// TIA Portal V18 export
FUNCTION "Controls" : Void   // FC8, LAD
{ S7_Optimized_Access := 'TRUE' }
VERSION : 0.1
// stored: AutoNumber true, IsIECCheckEnabled false, SetENOAutomatically false, UDAEnableTagReadback false
BEGIN

REGION Network 1: Function selected
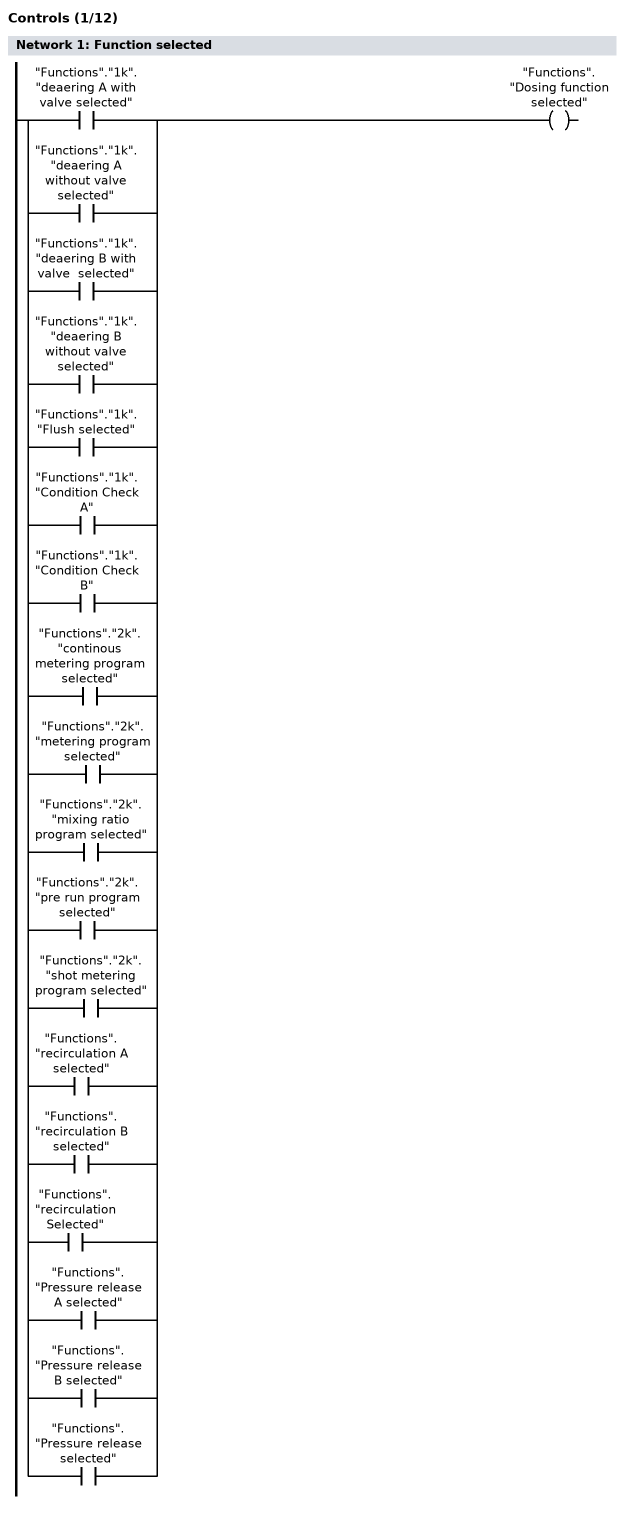
   RUNG wire#powerrail
      Contact( "Functions"."1k"."deaering A with valve selected" )
      wire#w1
      Coil( "Functions"."Dosing function selected" )
   END_RUNG
   RUNG wire#powerrail
      Contact( "Functions"."1k"."deaering A without valve selected" )
   END_RUNG wire#w1
   RUNG wire#powerrail
      Contact( "Functions"."1k"."deaering B with valve  selected" )
   END_RUNG wire#w1
   RUNG wire#powerrail
      Contact( "Functions"."1k"."deaering B without valve  selected" )
   END_RUNG wire#w1
   RUNG wire#powerrail
      Contact( "Functions"."1k"."Flush selected" )
   END_RUNG wire#w1
   RUNG wire#powerrail
      Contact( "Functions"."1k"."Condition Check A" )
   END_RUNG wire#w1
   RUNG wire#powerrail
      Contact( "Functions"."1k"."Condition Check B" )
   END_RUNG wire#w1
   RUNG wire#powerrail
      Contact( "Functions"."2k"."continous metering program selected" )
   END_RUNG wire#w1
   RUNG wire#powerrail
      Contact( "Functions"."2k"."metering program selected" )
   END_RUNG wire#w1
   RUNG wire#powerrail
      Contact( "Functions"."2k"."mixing ratio program selected" )
   END_RUNG wire#w1
   RUNG wire#powerrail
      Contact( "Functions"."2k"."pre run program selected" )
   END_RUNG wire#w1
   RUNG wire#powerrail
      Contact( "Functions"."2k"."shot metering program selected" )
   END_RUNG wire#w1
   RUNG wire#powerrail
      Contact( "Functions"."recirculation A selected" )
   END_RUNG wire#w1
   RUNG wire#powerrail
      Contact( "Functions"."recirculation B selected" )
   END_RUNG wire#w1
   RUNG wire#powerrail
      Contact( "Functions"."recirculation Selected" )
   END_RUNG wire#w1
   RUNG wire#powerrail
      Contact( "Functions"."Pressure release A selected" )
   END_RUNG wire#w1
   RUNG wire#powerrail
      Contact( "Functions"."Pressure release B selected" )
   END_RUNG wire#w1
   RUNG wire#powerrail
      Contact( "Functions"."Pressure release selected" )
   END_RUNG wire#w1
   // the same network as SCL:
   "Functions"."Dosing function selected" := "Functions"."1k"."deaering A with valve selected" OR "Functions"."1k"."deaering A without valve selected" OR "Functions"."1k"."deaering B with valve  selected" OR "Functions"."1k"."deaering B without valve  selected" OR "Functions"."1k"."Flush selected" OR "Functions"."1k"."Condition Check A" OR "Functions"."1k"."Condition Check B" OR "Functions"."2k"."continous metering program selected" OR "Functions"."2k"."metering program selected" OR "Functions"."2k"."mixing ratio program selected" OR "Functions"."2k"."pre run program selected" OR "Functions"."2k"."shot metering program selected" OR "Functions"."recirculation A selected" OR "Functions"."recirculation B selected" OR "Functions"."recirculation Selected" OR "Functions"."Pressure release A selected" OR "Functions"."Pressure release B selected" OR "Functions"."Pressure release selected";
END_REGION

REGION Network 2: Deselect all function
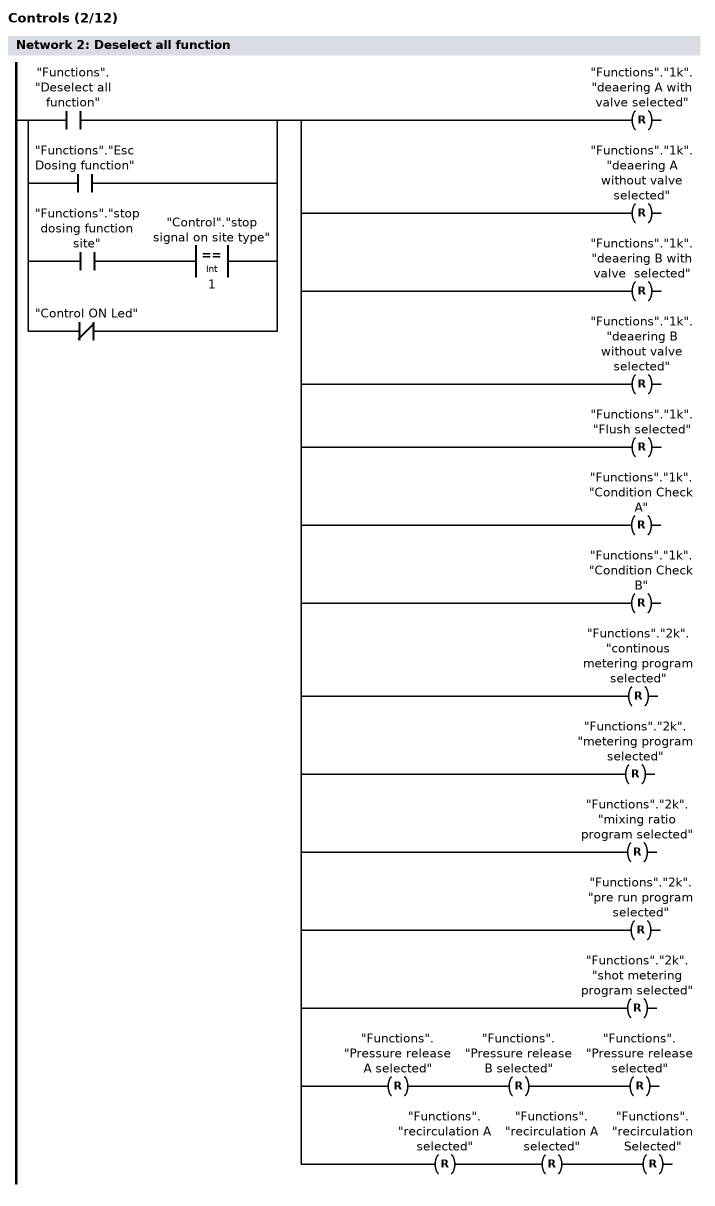
   RUNG wire#powerrail
      Contact( "Functions"."Deselect all function" )
      wire#w1
      R_Coil( "Functions"."1k"."deaering A with valve selected" )
   END_RUNG
   RUNG wire#powerrail
      Contact( "Functions"."Esc Dosing function" )
   END_RUNG wire#w1
   RUNG wire#powerrail
      Contact( "Functions"."stop dosing function site" )
      { S7_Templates := "SrcType := Int" } EQ_Contact(in1 := "Control"."stop signal on site type", in2 := 1)
   END_RUNG wire#w1
   RUNG wire#powerrail
      I_Contact( "Control ON Led" )
   END_RUNG wire#w1
   RUNG wire#w1
      R_Coil( "Functions"."1k"."deaering A without valve selected" )
   END_RUNG
   RUNG wire#w1
      R_Coil( "Functions"."1k"."deaering B with valve  selected" )
   END_RUNG
   RUNG wire#w1
      R_Coil( "Functions"."1k"."deaering B without valve  selected" )
   END_RUNG
   RUNG wire#w1
      R_Coil( "Functions"."1k"."Flush selected" )
   END_RUNG
   RUNG wire#w1
      R_Coil( "Functions"."1k"."Condition Check A" )
   END_RUNG
   RUNG wire#w1
      R_Coil( "Functions"."1k"."Condition Check B" )
   END_RUNG
   RUNG wire#w1
      R_Coil( "Functions"."2k"."continous metering program selected" )
   END_RUNG
   RUNG wire#w1
      R_Coil( "Functions"."2k"."metering program selected" )
   END_RUNG
   RUNG wire#w1
      R_Coil( "Functions"."2k"."mixing ratio program selected" )
   END_RUNG
   RUNG wire#w1
      R_Coil( "Functions"."2k"."pre run program selected" )
   END_RUNG
   RUNG wire#w1
      R_Coil( "Functions"."2k"."shot metering program selected" )
   END_RUNG
   RUNG wire#w1
      R_Coil( "Functions"."Pressure release A selected" )
      R_Coil( "Functions"."Pressure release B selected" )
      R_Coil( "Functions"."Pressure release selected" )
   END_RUNG
   RUNG wire#w1
      R_Coil( "Functions"."recirculation A selected" )
      R_Coil( "Functions"."recirculation A selected" )
      R_Coil( "Functions"."recirculation Selected" )
   END_RUNG
   // the same network as SCL:
   IF "Functions"."Deselect all function" OR "Functions"."Esc Dosing function" OR ("Functions"."stop dosing function site" AND ("Control"."stop signal on site type" = 1)) OR NOT "Control ON Led" THEN
       "Functions"."1k"."deaering A with valve selected" := FALSE;
       "Functions"."1k"."deaering A without valve selected" := FALSE;
       "Functions"."1k"."deaering B with valve  selected" := FALSE;
       "Functions"."1k"."deaering B without valve  selected" := FALSE;
       "Functions"."1k"."Flush selected" := FALSE;
       "Functions"."1k"."Condition Check A" := FALSE;
       "Functions"."1k"."Condition Check B" := FALSE;
       "Functions"."2k"."continous metering program selected" := FALSE;
       "Functions"."2k"."metering program selected" := FALSE;
       "Functions"."2k"."mixing ratio program selected" := FALSE;
       "Functions"."2k"."pre run program selected" := FALSE;
       "Functions"."2k"."shot metering program selected" := FALSE;
       "Functions"."Pressure release A selected" := FALSE;
       "Functions"."Pressure release B selected" := FALSE;
       "Functions"."Pressure release selected" := FALSE;
       "Functions"."recirculation A selected" := FALSE;
       "Functions"."recirculation A selected" := FALSE;
       "Functions"."recirculation Selected" := FALSE;
   END_IF;
END_REGION

REGION Network 3: Deselect all function During Refilling
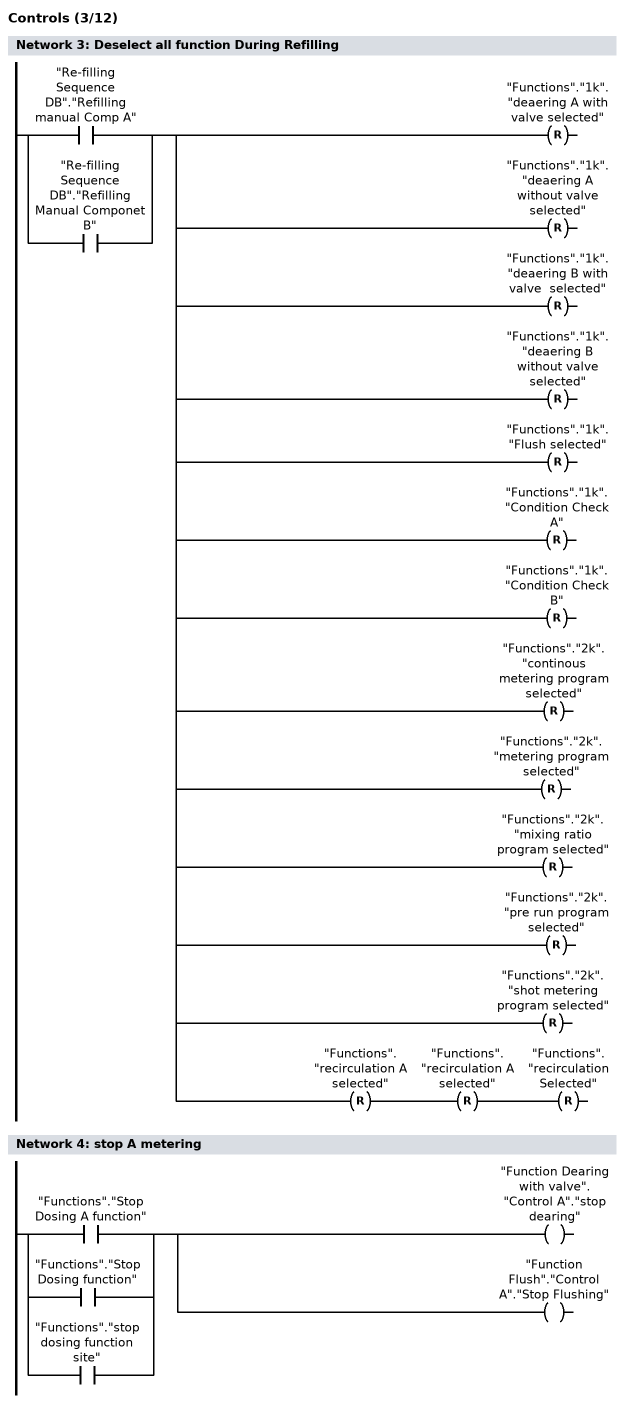
   RUNG wire#powerrail
      Contact( "Re-filling Sequence DB"."Refilling manual Comp A" )
      wire#w1
      R_Coil( "Functions"."1k"."deaering A with valve selected" )
   END_RUNG
   RUNG wire#powerrail
      Contact( "Re-filling Sequence DB"."Refilling Manual Componet B" )
   END_RUNG wire#w1
   RUNG wire#w1
      R_Coil( "Functions"."1k"."deaering A without valve selected" )
   END_RUNG
   RUNG wire#w1
      R_Coil( "Functions"."1k"."deaering B with valve  selected" )
   END_RUNG
   RUNG wire#w1
      R_Coil( "Functions"."1k"."deaering B without valve  selected" )
   END_RUNG
   RUNG wire#w1
      R_Coil( "Functions"."1k"."Flush selected" )
   END_RUNG
   RUNG wire#w1
      R_Coil( "Functions"."1k"."Condition Check A" )
   END_RUNG
   RUNG wire#w1
      R_Coil( "Functions"."1k"."Condition Check B" )
   END_RUNG
   RUNG wire#w1
      R_Coil( "Functions"."2k"."continous metering program selected" )
   END_RUNG
   RUNG wire#w1
      R_Coil( "Functions"."2k"."metering program selected" )
   END_RUNG
   RUNG wire#w1
      R_Coil( "Functions"."2k"."mixing ratio program selected" )
   END_RUNG
   RUNG wire#w1
      R_Coil( "Functions"."2k"."pre run program selected" )
   END_RUNG
   RUNG wire#w1
      R_Coil( "Functions"."2k"."shot metering program selected" )
   END_RUNG
   RUNG wire#w1
      R_Coil( "Functions"."recirculation A selected" )
      R_Coil( "Functions"."recirculation A selected" )
      R_Coil( "Functions"."recirculation Selected" )
   END_RUNG
   // the same network as SCL:
   IF "Re-filling Sequence DB"."Refilling manual Comp A" OR "Re-filling Sequence DB"."Refilling Manual Componet B" THEN
       "Functions"."1k"."deaering A with valve selected" := FALSE;
       "Functions"."1k"."deaering A without valve selected" := FALSE;
       "Functions"."1k"."deaering B with valve  selected" := FALSE;
       "Functions"."1k"."deaering B without valve  selected" := FALSE;
       "Functions"."1k"."Flush selected" := FALSE;
       "Functions"."1k"."Condition Check A" := FALSE;
       "Functions"."1k"."Condition Check B" := FALSE;
       "Functions"."2k"."continous metering program selected" := FALSE;
       "Functions"."2k"."metering program selected" := FALSE;
       "Functions"."2k"."mixing ratio program selected" := FALSE;
       "Functions"."2k"."pre run program selected" := FALSE;
       "Functions"."2k"."shot metering program selected" := FALSE;
       "Functions"."recirculation A selected" := FALSE;
       "Functions"."recirculation A selected" := FALSE;
       "Functions"."recirculation Selected" := FALSE;
   END_IF;
END_REGION

REGION Network 4: stop A metering
   RUNG wire#powerrail
      Contact( "Functions"."Stop Dosing A function" )
      wire#w1
      Coil( "Function Dearing with valve"."Control A"."stop dearing" )
   END_RUNG
   RUNG wire#powerrail
      Contact( "Functions"."Stop Dosing function" )
   END_RUNG wire#w1
   RUNG wire#powerrail
      Contact( "Functions"."stop dosing function site" )
   END_RUNG wire#w1
   RUNG wire#w1
      Coil( "Function Flush"."Control A"."Stop Flushing" )
   END_RUNG
   // the same network as SCL:
   "Function Dearing with valve"."Control A"."stop dearing" := "Functions"."Stop Dosing A function" OR "Functions"."Stop Dosing function" OR "Functions"."stop dosing function site";
   "Function Flush"."Control A"."Stop Flushing" := "Function Dearing with valve"."Control A"."stop dearing";
END_REGION

REGION Network 5: stop B metering
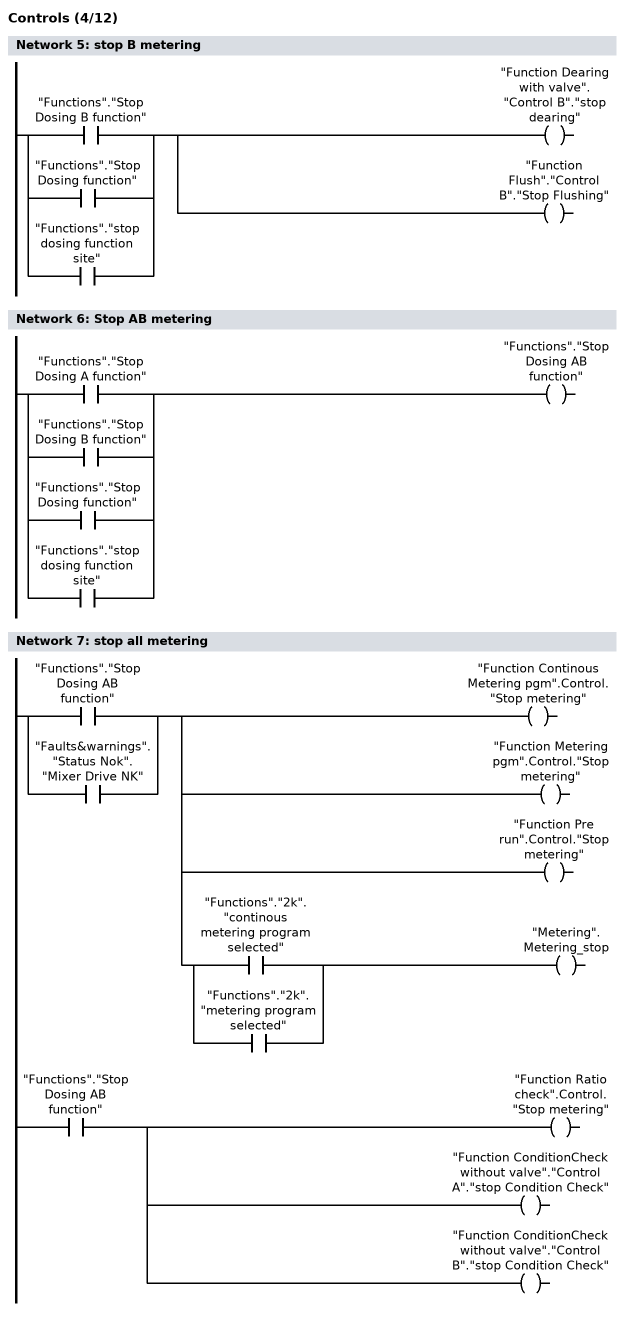
   RUNG wire#powerrail
      Contact( "Functions"."Stop Dosing B function" )
      wire#w1
      Coil( "Function Dearing with valve"."Control B"."stop dearing" )
   END_RUNG
   RUNG wire#powerrail
      Contact( "Functions"."Stop Dosing function" )
   END_RUNG wire#w1
   RUNG wire#powerrail
      Contact( "Functions"."stop dosing function site" )
   END_RUNG wire#w1
   RUNG wire#w1
      Coil( "Function Flush"."Control B"."Stop Flushing" )
   END_RUNG
   // the same network as SCL:
   "Function Dearing with valve"."Control B"."stop dearing" := "Functions"."Stop Dosing B function" OR "Functions"."Stop Dosing function" OR "Functions"."stop dosing function site";
   "Function Flush"."Control B"."Stop Flushing" := "Function Dearing with valve"."Control B"."stop dearing";
END_REGION

REGION Network 6: Stop AB metering
   RUNG wire#powerrail
      Contact( "Functions"."Stop Dosing A function" )
      wire#w1
      Coil( "Functions"."Stop Dosing AB function" )
   END_RUNG
   RUNG wire#powerrail
      Contact( "Functions"."Stop Dosing B function" )
   END_RUNG wire#w1
   RUNG wire#powerrail
      Contact( "Functions"."Stop Dosing function" )
   END_RUNG wire#w1
   RUNG wire#powerrail
      Contact( "Functions"."stop dosing function site" )
   END_RUNG wire#w1
   // the same network as SCL:
   "Functions"."Stop Dosing AB function" := "Functions"."Stop Dosing A function" OR "Functions"."Stop Dosing B function" OR "Functions"."Stop Dosing function" OR "Functions"."stop dosing function site";
END_REGION

REGION Network 7: stop all metering
   RUNG wire#powerrail
      Contact( "Functions"."Stop Dosing AB function" )
      wire#w1
      Coil( "Function Continous Metering pgm".Control."Stop metering" )
   END_RUNG
   RUNG wire#powerrail
      Contact( "Faults&warnings"."Status Nok"."Mixer Drive NK" )
   END_RUNG wire#w1
   RUNG wire#w1
      Coil( "Function Metering pgm".Control."Stop metering" )
   END_RUNG
   RUNG wire#w1
      Coil( "Function Pre run".Control."Stop metering" )
   END_RUNG
   RUNG wire#w1
      Contact( "Functions"."2k"."continous metering program selected" )
      wire#w2
      Coil( "Metering".Metering_stop )
   END_RUNG
   RUNG wire#w1
      Contact( "Functions"."2k"."metering program selected" )
   END_RUNG wire#w2
   RUNG wire#powerrail
      Contact( "Functions"."Stop Dosing AB function" )
      wire#w3
      Coil( "Function Ratio check".Control."Stop metering" )
   END_RUNG
   RUNG wire#w3
      Coil( "Function ConditionCheck without valve"."Control A"."stop Condition Check" )
   END_RUNG
   RUNG wire#w3
      Coil( "Function ConditionCheck without valve"."Control B"."stop Condition Check" )
   END_RUNG
   // the same network as SCL:
   "Function Continous Metering pgm".Control."Stop metering" := "Functions"."Stop Dosing AB function" OR "Faults&warnings"."Status Nok"."Mixer Drive NK";
   "Function Metering pgm".Control."Stop metering" := "Function Continous Metering pgm".Control."Stop metering";
   "Function Pre run".Control."Stop metering" := "Function Continous Metering pgm".Control."Stop metering";
   "Metering".Metering_stop := "Function Continous Metering pgm".Control."Stop metering" AND ("Functions"."2k"."continous metering program selected" OR "Functions"."2k"."metering program selected");
   "Function Ratio check".Control."Stop metering" := "Functions"."Stop Dosing AB function";
   "Function ConditionCheck without valve"."Control A"."stop Condition Check" := "Functions"."Stop Dosing AB function";
   "Function ConditionCheck without valve"."Control B"."stop Condition Check" := "Functions"."Stop Dosing AB function";
END_REGION

REGION Network 8: Critical fault Block A metering
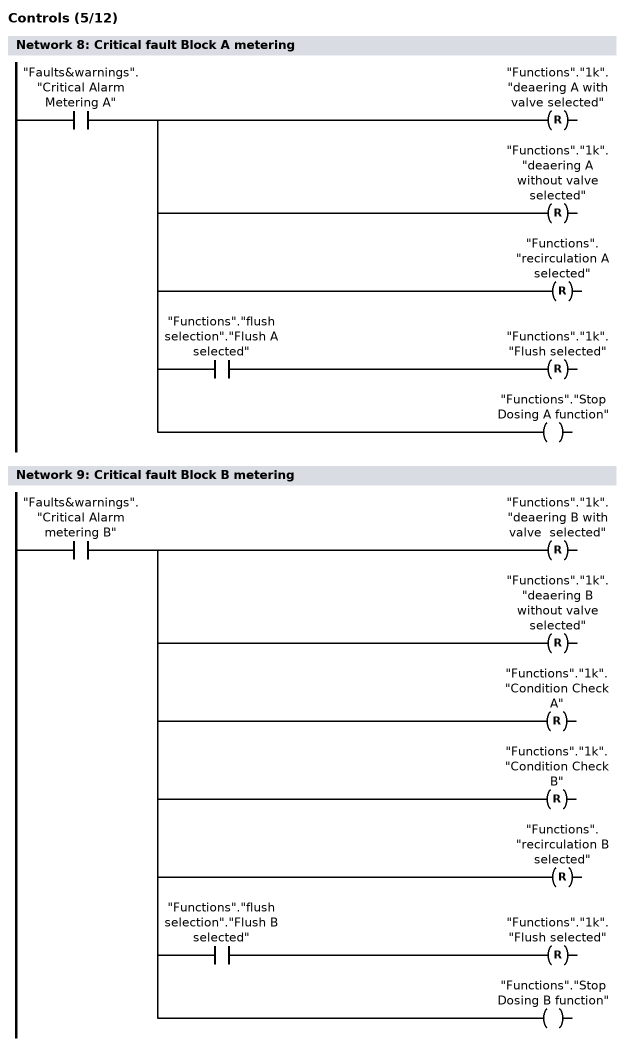
   RUNG wire#powerrail
      Contact( "Faults&warnings"."Critical Alarm Metering A" )
      wire#w1
      R_Coil( "Functions"."1k"."deaering A with valve selected" )
   END_RUNG
   RUNG wire#w1
      R_Coil( "Functions"."1k"."deaering A without valve selected" )
   END_RUNG
   RUNG wire#w1
      R_Coil( "Functions"."recirculation A selected" )
   END_RUNG
   RUNG wire#w1
      Contact( "Functions"."flush selection"."Flush A selected" )
      R_Coil( "Functions"."1k"."Flush selected" )
   END_RUNG
   RUNG wire#w1
      Coil( "Functions"."Stop Dosing A function" )
   END_RUNG
   // the same network as SCL:
   IF "Faults&warnings"."Critical Alarm Metering A" THEN
       "Functions"."1k"."deaering A with valve selected" := FALSE;
       "Functions"."1k"."deaering A without valve selected" := FALSE;
       "Functions"."recirculation A selected" := FALSE;
   END_IF;
   IF "Faults&warnings"."Critical Alarm Metering A" AND "Functions"."flush selection"."Flush A selected" THEN
       "Functions"."1k"."Flush selected" := FALSE;
   END_IF;
   "Functions"."Stop Dosing A function" := "Faults&warnings"."Critical Alarm Metering A";
END_REGION

REGION Network 9: Critical fault Block B metering
   RUNG wire#powerrail
      Contact( "Faults&warnings"."Critical Alarm metering B" )
      wire#w1
      R_Coil( "Functions"."1k"."deaering B with valve  selected" )
   END_RUNG
   RUNG wire#w1
      R_Coil( "Functions"."1k"."deaering B without valve  selected" )
   END_RUNG
   RUNG wire#w1
      R_Coil( "Functions"."1k"."Condition Check A" )
   END_RUNG
   RUNG wire#w1
      R_Coil( "Functions"."1k"."Condition Check B" )
   END_RUNG
   RUNG wire#w1
      R_Coil( "Functions"."recirculation B selected" )
   END_RUNG
   RUNG wire#w1
      Contact( "Functions"."flush selection"."Flush B selected" )
      R_Coil( "Functions"."1k"."Flush selected" )
   END_RUNG
   RUNG wire#w1
      Coil( "Functions"."Stop Dosing B function" )
   END_RUNG
   // the same network as SCL:
   IF "Faults&warnings"."Critical Alarm metering B" THEN
       "Functions"."1k"."deaering B with valve  selected" := FALSE;
       "Functions"."1k"."deaering B without valve  selected" := FALSE;
       "Functions"."1k"."Condition Check A" := FALSE;
       "Functions"."1k"."Condition Check B" := FALSE;
       "Functions"."recirculation B selected" := FALSE;
   END_IF;
   IF "Faults&warnings"."Critical Alarm metering B" AND "Functions"."flush selection"."Flush B selected" THEN
       "Functions"."1k"."Flush selected" := FALSE;
   END_IF;
   "Functions"."Stop Dosing B function" := "Faults&warnings"."Critical Alarm metering B";
END_REGION

REGION Network 10: Critical fault block all metering
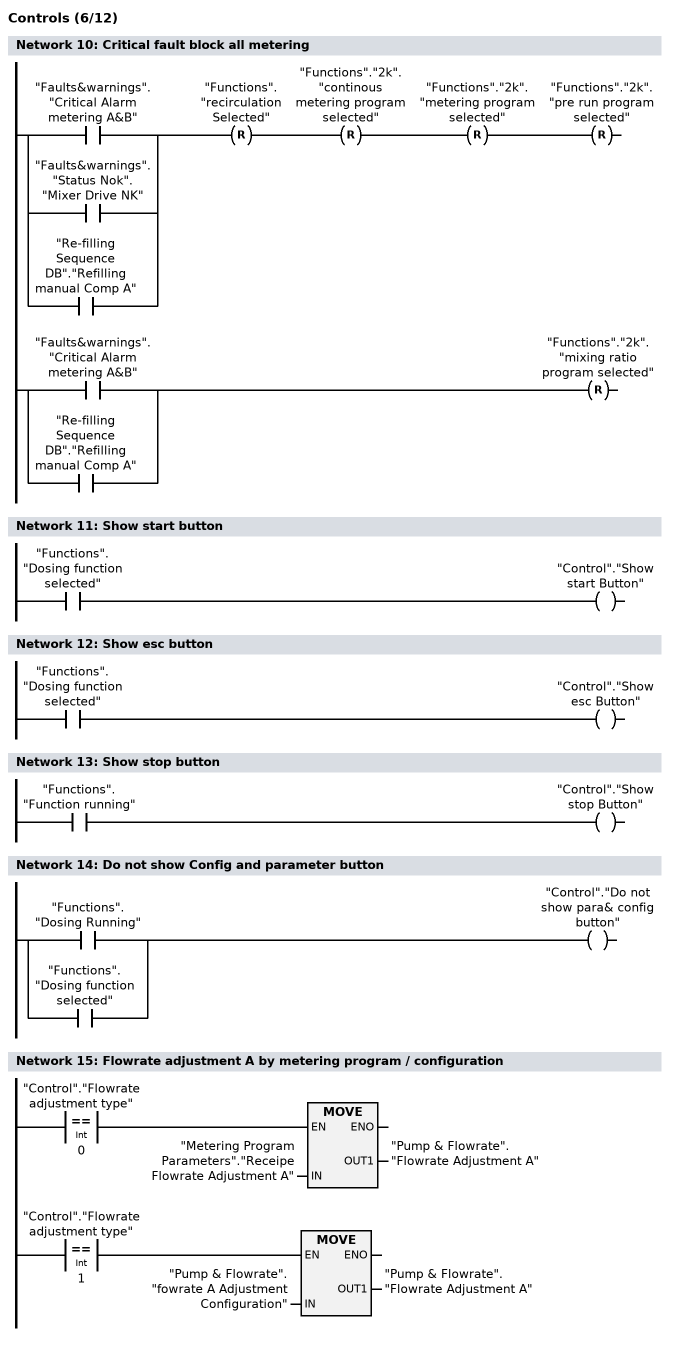
   RUNG wire#powerrail
      Contact( "Faults&warnings"."Critical Alarm metering A&B" )
      wire#w1
      R_Coil( "Functions"."recirculation Selected" )
      R_Coil( "Functions"."2k"."continous metering program selected" )
      R_Coil( "Functions"."2k"."metering program selected" )
      R_Coil( "Functions"."2k"."pre run program selected" )
   END_RUNG
   RUNG wire#powerrail
      Contact( "Faults&warnings"."Status Nok"."Mixer Drive NK" )
   END_RUNG wire#w1
   RUNG wire#powerrail
      Contact( "Re-filling Sequence DB"."Refilling manual Comp A" )
   END_RUNG wire#w1
   RUNG wire#powerrail
      Contact( "Faults&warnings"."Critical Alarm metering A&B" )
      wire#w2
      R_Coil( "Functions"."2k"."mixing ratio program selected" )
   END_RUNG
   RUNG wire#powerrail
      Contact( "Re-filling Sequence DB"."Refilling manual Comp A" )
   END_RUNG wire#w2
   // the same network as SCL:
   IF "Faults&warnings"."Critical Alarm metering A&B" OR "Faults&warnings"."Status Nok"."Mixer Drive NK" OR "Re-filling Sequence DB"."Refilling manual Comp A" THEN
       "Functions"."recirculation Selected" := FALSE;
       "Functions"."2k"."continous metering program selected" := FALSE;
       "Functions"."2k"."metering program selected" := FALSE;
       "Functions"."2k"."pre run program selected" := FALSE;
   END_IF;
   IF "Faults&warnings"."Critical Alarm metering A&B" OR "Re-filling Sequence DB"."Refilling manual Comp A" THEN
       "Functions"."2k"."mixing ratio program selected" := FALSE;
   END_IF;
END_REGION

REGION Network 11: Show start button
   RUNG wire#powerrail
      Contact( "Functions"."Dosing function selected" )
      Coil( "Control"."Show start Button" )
   END_RUNG
   // the same network as SCL:
   "Control"."Show start Button" := "Functions"."Dosing function selected";
END_REGION

REGION Network 12: Show esc button
   RUNG wire#powerrail
      Contact( "Functions"."Dosing function selected" )
      Coil( "Control"."Show esc Button" )
   END_RUNG
   // the same network as SCL:
   "Control"."Show esc Button" := "Functions"."Dosing function selected";
END_REGION

REGION Network 13: Show stop button
   RUNG wire#powerrail
      Contact( "Functions"."Function running" )
      Coil( "Control"."Show stop Button" )
   END_RUNG
   // the same network as SCL:
   "Control"."Show stop Button" := "Functions"."Function running";
END_REGION

REGION Network 14: Do not show Config and parameter button
   RUNG wire#powerrail
      Contact( "Functions"."Dosing Running" )
      wire#w1
      Coil( "Control"."Do not show para& config button" )
   END_RUNG
   RUNG wire#powerrail
      Contact( "Functions"."Dosing function selected" )
   END_RUNG wire#w1
   // the same network as SCL:
   "Control"."Do not show para& config button" := "Functions"."Dosing Running" OR "Functions"."Dosing function selected";
END_REGION

REGION Network 15: Flowrate adjustment A by metering program / configuration
   IF "Control"."Flowrate adjustment type" = 0 THEN
       "Pump & Flowrate"."Flowrate Adjustment A" := "Metering Program Parameters"."Receipe Flowrate Adjustment A";
   END_IF;
   IF "Control"."Flowrate adjustment type" = 1 THEN
       "Pump & Flowrate"."Flowrate Adjustment A" := "Pump & Flowrate"."fowrate A Adjustment Configuration";
   END_IF;
END_REGION

REGION Network 16: Flowrate adjustment B by metering program / configuration
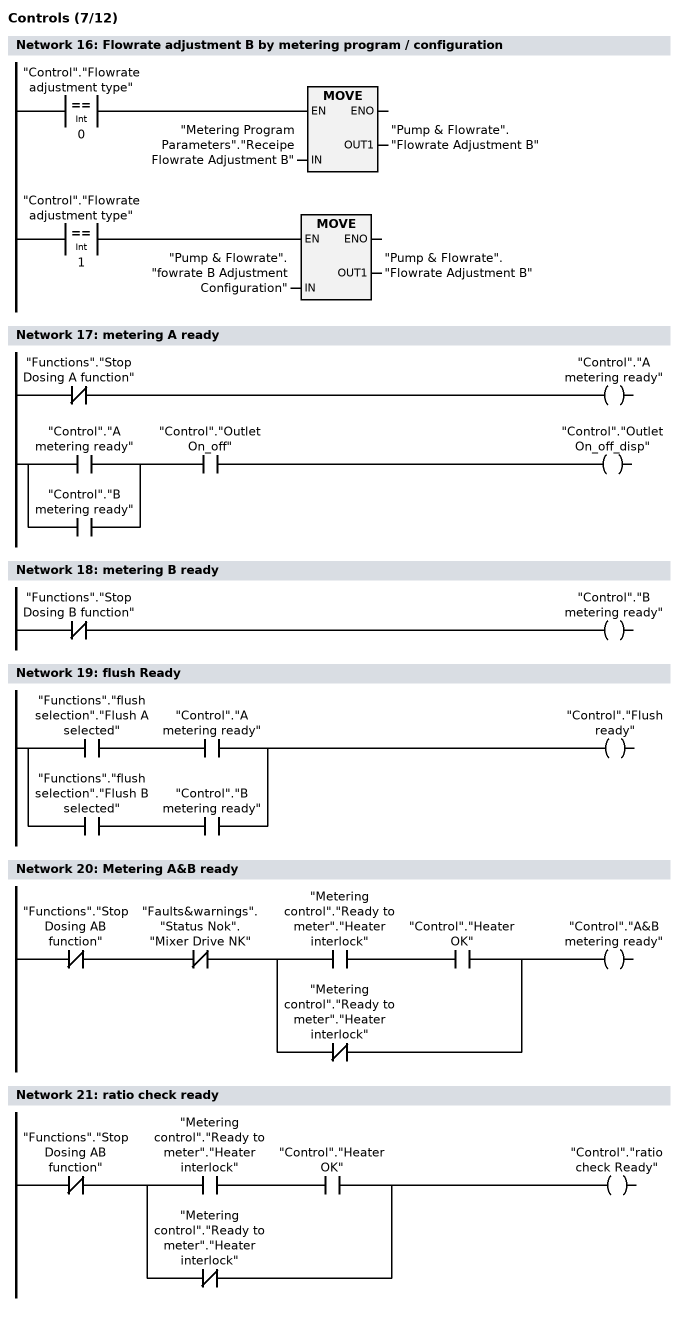
   IF "Control"."Flowrate adjustment type" = 0 THEN
       "Pump & Flowrate"."Flowrate Adjustment B" := "Metering Program Parameters"."Receipe Flowrate Adjustment B";
   END_IF;
   IF "Control"."Flowrate adjustment type" = 1 THEN
       "Pump & Flowrate"."Flowrate Adjustment B" := "Pump & Flowrate"."fowrate B Adjustment Configuration";
   END_IF;
END_REGION

REGION Network 17: metering A ready
   RUNG wire#powerrail
      I_Contact( "Functions"."Stop Dosing A function" )
      Coil( "Control"."A metering ready" )
   END_RUNG
   RUNG wire#powerrail
      Contact( "Control"."A metering ready" )
      wire#w1
      Contact( "Control"."Outlet On_off" )
      Coil( "Control"."Outlet On_off_disp" )
   END_RUNG
   RUNG wire#powerrail
      Contact( "Control"."B metering ready" )
   END_RUNG wire#w1
   // the same network as SCL:
   "Control"."A metering ready" := NOT "Functions"."Stop Dosing A function";
   "Control"."Outlet On_off_disp" := ("Control"."A metering ready" OR "Control"."B metering ready") AND "Control"."Outlet On_off";
END_REGION

REGION Network 18: metering B ready
   RUNG wire#powerrail
      I_Contact( "Functions"."Stop Dosing B function" )
      Coil( "Control"."B metering ready" )
   END_RUNG
   // the same network as SCL:
   "Control"."B metering ready" := NOT "Functions"."Stop Dosing B function";
END_REGION

REGION Network 19: flush Ready
   RUNG wire#powerrail
      Contact( "Functions"."flush selection"."Flush A selected" )
      Contact( "Control"."A metering ready" )
      wire#w1
      Coil( "Control"."Flush ready" )
   END_RUNG
   RUNG wire#powerrail
      Contact( "Functions"."flush selection"."Flush B selected" )
      Contact( "Control"."B metering ready" )
   END_RUNG wire#w1
   // the same network as SCL:
   "Control"."Flush ready" := ("Functions"."flush selection"."Flush A selected" AND "Control"."A metering ready") OR ("Functions"."flush selection"."Flush B selected" AND "Control"."B metering ready");
END_REGION

REGION Network 20: Metering A&B ready
   RUNG wire#powerrail
      I_Contact( "Functions"."Stop Dosing AB function" )
      I_Contact( "Faults&warnings"."Status Nok"."Mixer Drive NK" )
      wire#w1
      Contact( "Metering control"."Ready to meter"."Heater interlock" )
      Contact( "Control"."Heater OK" )
      wire#w2
      Coil( "Control"."A&B metering ready" )
   END_RUNG
   RUNG wire#w1
      I_Contact( "Metering control"."Ready to meter"."Heater interlock" )
   END_RUNG wire#w2
   // the same network as SCL:
   "Control"."A&B metering ready" := NOT "Functions"."Stop Dosing AB function" AND NOT "Faults&warnings"."Status Nok"."Mixer Drive NK" AND (("Metering control"."Ready to meter"."Heater interlock" AND "Control"."Heater OK") OR NOT "Metering control"."Ready to meter"."Heater interlock");
END_REGION

REGION Network 21: ratio check ready
   RUNG wire#powerrail
      I_Contact( "Functions"."Stop Dosing AB function" )
      wire#w1
      Contact( "Metering control"."Ready to meter"."Heater interlock" )
      Contact( "Control"."Heater OK" )
      wire#w2
      Coil( "Control"."ratio check Ready" )
   END_RUNG
   RUNG wire#w1
      I_Contact( "Metering control"."Ready to meter"."Heater interlock" )
   END_RUNG wire#w2
   // the same network as SCL:
   "Control"."ratio check Ready" := NOT "Functions"."Stop Dosing AB function" AND (("Metering control"."Ready to meter"."Heater interlock" AND "Control"."Heater OK") OR NOT "Metering control"."Ready to meter"."Heater interlock");
END_REGION

REGION Network 22: Metering program ready
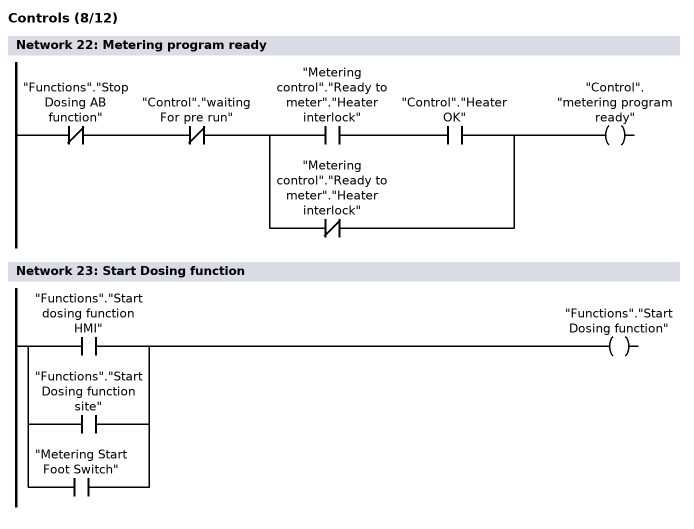
   RUNG wire#powerrail
      I_Contact( "Functions"."Stop Dosing AB function" )
      I_Contact( "Control"."waiting For pre run" )
      wire#w1
      Contact( "Metering control"."Ready to meter"."Heater interlock" )
      Contact( "Control"."Heater OK" )
      wire#w2
      Coil( "Control"."metering program ready" )
   END_RUNG
   RUNG wire#w1
      I_Contact( "Metering control"."Ready to meter"."Heater interlock" )
   END_RUNG wire#w2
   // the same network as SCL:
   "Control"."metering program ready" := NOT "Functions"."Stop Dosing AB function" AND NOT "Control"."waiting For pre run" AND (("Metering control"."Ready to meter"."Heater interlock" AND "Control"."Heater OK") OR NOT "Metering control"."Ready to meter"."Heater interlock");
END_REGION

REGION Network 23: Start Dosing function
   RUNG wire#powerrail
      Contact( "Functions"."Start dosing function HMI" )
      wire#w1
      Coil( "Functions"."Start Dosing function" )
   END_RUNG
   RUNG wire#powerrail
      Contact( "Functions"."Start Dosing function site" )
   END_RUNG wire#w1
   RUNG wire#powerrail
      Contact( "Metering Start Foot Switch" )
   END_RUNG wire#w1
   // the same network as SCL:
   "Functions"."Start Dosing function" := "Functions"."Start dosing function HMI" OR "Functions"."Start Dosing function site" OR "Metering Start Foot Switch";
END_REGION

REGION Network 24: Dosing running
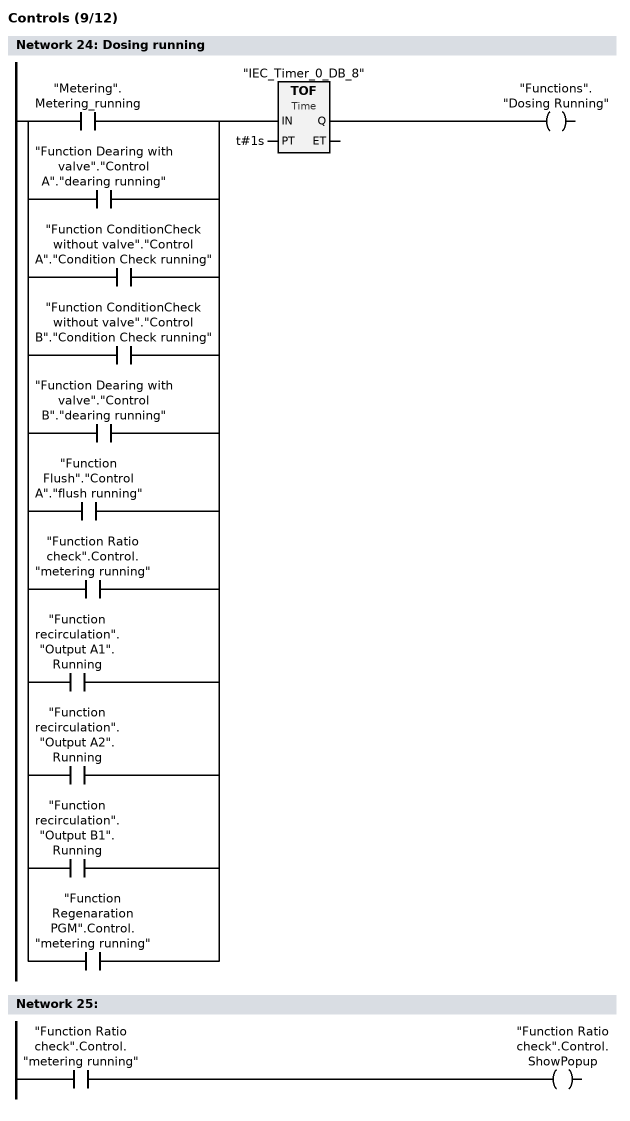
   RUNG wire#powerrail
      Contact( "Metering".Metering_running )
      wire#w1
      { S7_Templates := "time_type := Time" } "IEC_Timer_0_DB_8".TOF(pt := t#1s, et =>)
      Coil( "Functions"."Dosing Running" )
   END_RUNG
   RUNG wire#powerrail
      Contact( "Function Dearing with valve"."Control A"."dearing running" )
   END_RUNG wire#w1
   RUNG wire#powerrail
      Contact( "Function ConditionCheck without valve"."Control A"."Condition Check running" )
   END_RUNG wire#w1
   RUNG wire#powerrail
      Contact( "Function ConditionCheck without valve"."Control B"."Condition Check running" )
   END_RUNG wire#w1
   RUNG wire#powerrail
      Contact( "Function Dearing with valve"."Control B"."dearing running" )
   END_RUNG wire#w1
   RUNG wire#powerrail
      Contact( "Function Flush"."Control A"."flush running" )
   END_RUNG wire#w1
   RUNG wire#powerrail
      Contact( "Function Ratio check".Control."metering running" )
   END_RUNG wire#w1
   RUNG wire#powerrail
      Contact( "Function recirculation"."Output A1".Running )
   END_RUNG wire#w1
   RUNG wire#powerrail
      Contact( "Function recirculation"."Output A2".Running )
   END_RUNG wire#w1
   RUNG wire#powerrail
      Contact( "Function recirculation"."Output B1".Running )
   END_RUNG wire#w1
   RUNG wire#powerrail
      Contact( "Function Regenaration PGM".Control."metering running" )
   END_RUNG wire#w1
   // the same network as SCL:
   "IEC_Timer_0_DB_8".TOF(IN := "Metering".Metering_running OR "Function Dearing with valve"."Control A"."dearing running" OR "Function ConditionCheck without valve"."Control A"."Condition Check running" OR "Function ConditionCheck without valve"."Control B"."Condition Check running" OR "Function Dearing with valve"."Control B"."dearing running" OR "Function Flush"."Control A"."flush running" OR "Function Ratio check".Control."metering running" OR "Function recirculation"."Output A1".Running OR "Function recirculation"."Output A2".Running OR "Function recirculation"."Output B1".Running OR "Function Regenaration PGM".Control."metering running",
                          PT := t#1s);
   "Functions"."Dosing Running" := "IEC_Timer_0_DB_8".Q;
END_REGION

REGION Network 25
   RUNG wire#powerrail
      Contact( "Function Ratio check".Control."metering running" )
      Coil( "Function Ratio check".Control.ShowPopup )
   END_RUNG
   // the same network as SCL:
   "Function Ratio check".Control.ShowPopup := "Function Ratio check".Control."metering running";
END_REGION

REGION Network 26
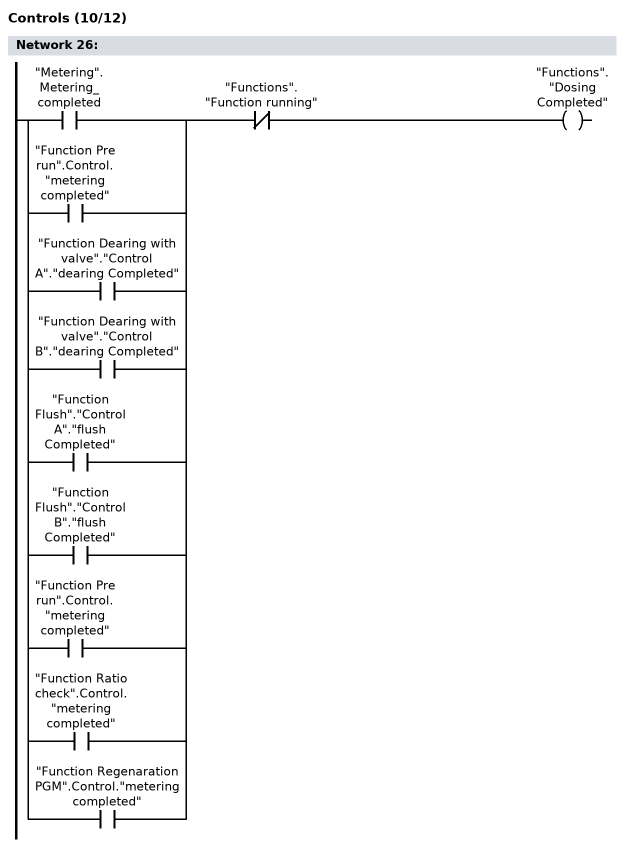
   RUNG wire#powerrail
      Contact( "Metering".Metering_completed )
      wire#w1
      I_Contact( "Functions"."Function running" )
      Coil( "Functions"."Dosing Completed" )
   END_RUNG
   RUNG wire#powerrail
      Contact( "Function Pre run".Control."metering completed" )
   END_RUNG wire#w1
   RUNG wire#powerrail
      Contact( "Function Dearing with valve"."Control A"."dearing Completed" )
   END_RUNG wire#w1
   RUNG wire#powerrail
      Contact( "Function Dearing with valve"."Control B"."dearing Completed" )
   END_RUNG wire#w1
   RUNG wire#powerrail
      Contact( "Function Flush"."Control A"."flush Completed" )
   END_RUNG wire#w1
   RUNG wire#powerrail
      Contact( "Function Flush"."Control B"."flush Completed" )
   END_RUNG wire#w1
   RUNG wire#powerrail
      Contact( "Function Pre run".Control."metering completed" )
   END_RUNG wire#w1
   RUNG wire#powerrail
      Contact( "Function Ratio check".Control."metering completed" )
   END_RUNG wire#w1
   RUNG wire#powerrail
      Contact( "Function Regenaration PGM".Control."metering completed" )
   END_RUNG wire#w1
   // the same network as SCL:
   "Functions"."Dosing Completed" := ("Metering".Metering_completed OR "Function Pre run".Control."metering completed" OR "Function Dearing with valve"."Control A"."dearing Completed" OR "Function Dearing with valve"."Control B"."dearing Completed" OR "Function Flush"."Control A"."flush Completed" OR "Function Flush"."Control B"."flush Completed" OR "Function Pre run".Control."metering completed" OR "Function Ratio check".Control."metering completed" OR "Function Regenaration PGM".Control."metering completed") AND NOT "Functions"."Function running";
END_REGION

REGION Network 27: Function running
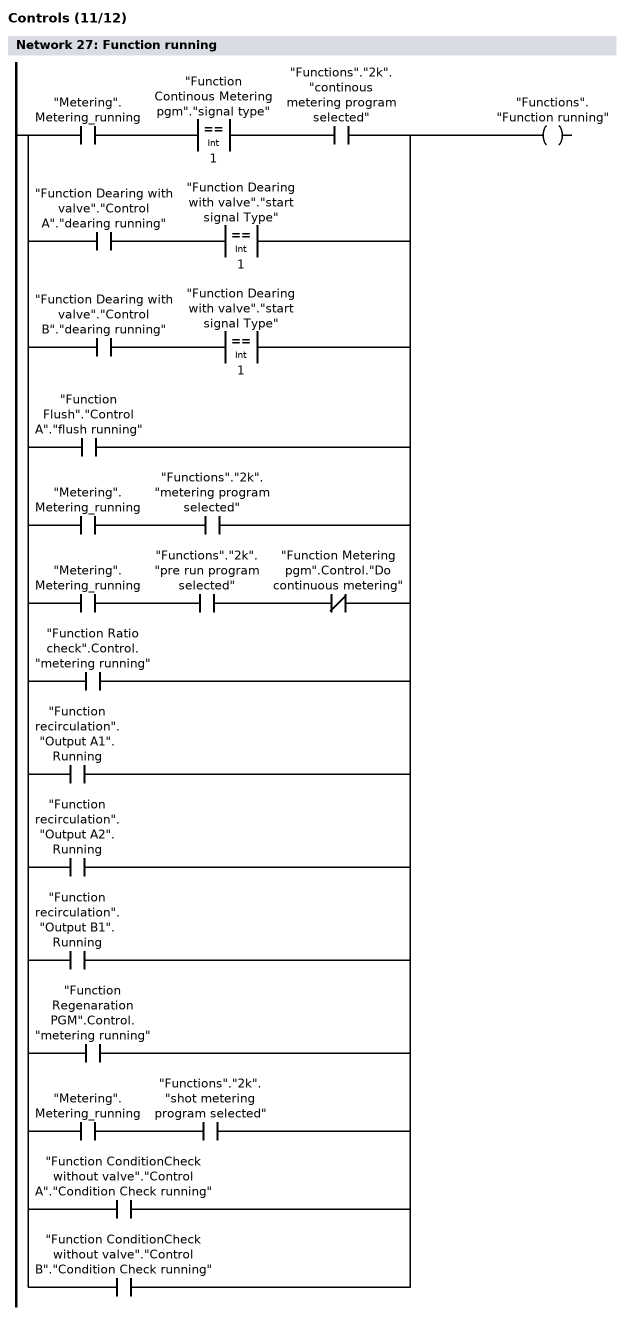
   RUNG wire#powerrail
      Contact( "Metering".Metering_running )
      { S7_Templates := "SrcType := Int" } EQ_Contact(in1 := "Function Continous Metering pgm"."signal type", in2 := 1)
      Contact( "Functions"."2k"."continous metering program selected" )
      wire#w1
      Coil( "Functions"."Function running" )
   END_RUNG
   RUNG wire#powerrail
      Contact( "Function Dearing with valve"."Control A"."dearing running" )
      { S7_Templates := "SrcType := Int" } EQ_Contact(in1 := "Function Dearing with valve"."start signal Type", in2 := 1)
   END_RUNG wire#w1
   RUNG wire#powerrail
      Contact( "Function Dearing with valve"."Control B"."dearing running" )
      { S7_Templates := "SrcType := Int" } EQ_Contact(in1 := "Function Dearing with valve"."start signal Type", in2 := 1)
   END_RUNG wire#w1
   RUNG wire#powerrail
      Contact( "Function Flush"."Control A"."flush running" )
   END_RUNG wire#w1
   RUNG wire#powerrail
      Contact( "Metering".Metering_running )
      Contact( "Functions"."2k"."metering program selected" )
   END_RUNG wire#w1
   RUNG wire#powerrail
      Contact( "Metering".Metering_running )
      Contact( "Functions"."2k"."pre run program selected" )
      I_Contact( "Function Metering pgm".Control."Do continuous metering" )
   END_RUNG wire#w1
   RUNG wire#powerrail
      Contact( "Function Ratio check".Control."metering running" )
   END_RUNG wire#w1
   RUNG wire#powerrail
      Contact( "Function recirculation"."Output A1".Running )
   END_RUNG wire#w1
   RUNG wire#powerrail
      Contact( "Function recirculation"."Output A2".Running )
   END_RUNG wire#w1
   RUNG wire#powerrail
      Contact( "Function recirculation"."Output B1".Running )
   END_RUNG wire#w1
   RUNG wire#powerrail
      Contact( "Function Regenaration PGM".Control."metering running" )
   END_RUNG wire#w1
   RUNG wire#powerrail
      Contact( "Metering".Metering_running )
      Contact( "Functions"."2k"."shot metering program selected" )
   END_RUNG wire#w1
   RUNG wire#powerrail
      Contact( "Function ConditionCheck without valve"."Control A"."Condition Check running" )
   END_RUNG wire#w1
   RUNG wire#powerrail
      Contact( "Function ConditionCheck without valve"."Control B"."Condition Check running" )
   END_RUNG wire#w1
   // the same network as SCL:
   "Functions"."Function running" := ("Metering".Metering_running AND ("Function Continous Metering pgm"."signal type" = 1) AND "Functions"."2k"."continous metering program selected") OR ("Function Dearing with valve"."Control A"."dearing running" AND ("Function Dearing with valve"."start signal Type" = 1)) OR ("Function Dearing with valve"."Control B"."dearing running" AND ("Function Dearing with valve"."start signal Type" = 1)) OR "Function Flush"."Control A"."flush running" OR ("Metering".Metering_running AND "Functions"."2k"."metering program selected") OR ("Metering".Metering_running AND "Functions"."2k"."pre run program selected" AND NOT "Function Metering pgm".Control."Do continuous metering") OR "Function Ratio check".Control."metering running" OR "Function recirculation"."Output A1".Running OR "Function recirculation"."Output A2".Running OR "Function recirculation"."Output B1".Running OR "Function Regenaration PGM".Control."metering running" OR ("Metering".Metering_running AND "Functions"."2k"."shot metering program selected") OR "Function ConditionCheck without valve"."Control A"."Condition Check running" OR "Function ConditionCheck without valve"."Control B"."Condition Check running";
END_REGION

REGION Network 28: show alarm textfield in all screen
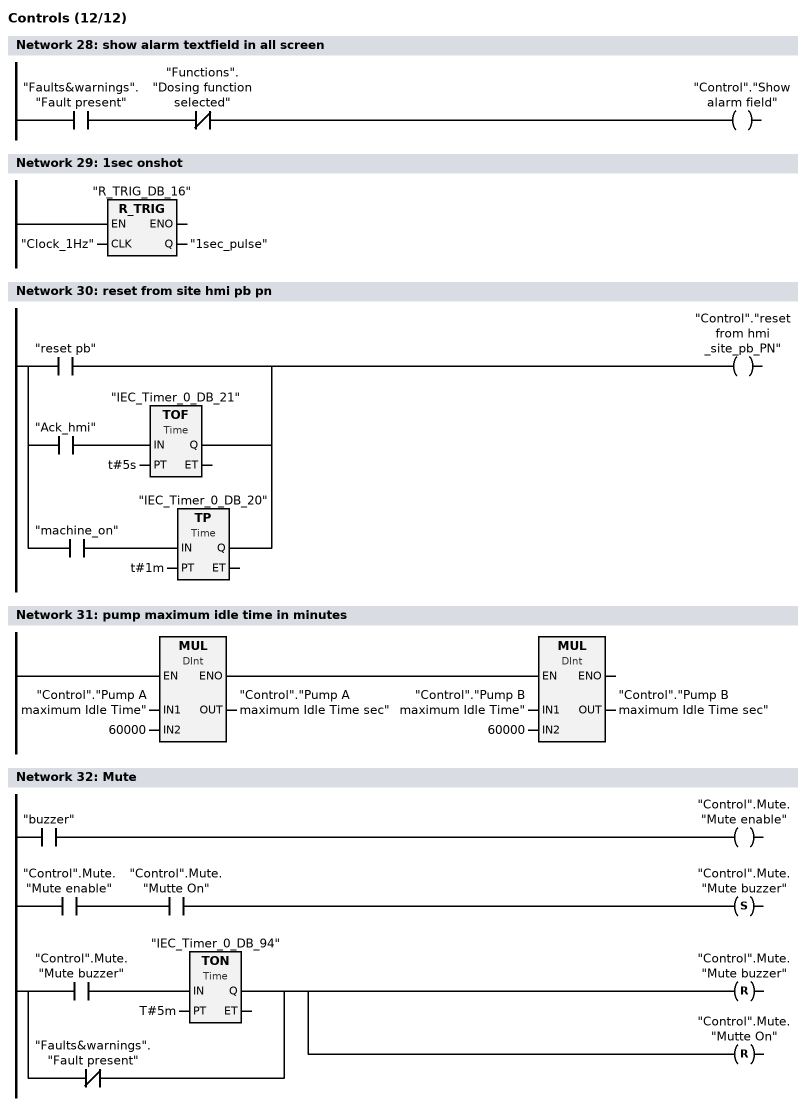
   RUNG wire#powerrail
      Contact( "Faults&warnings"."Fault present" )
      I_Contact( "Functions"."Dosing function selected" )
      Coil( "Control"."Show alarm field" )
   END_RUNG
   // the same network as SCL:
   "Control"."Show alarm field" := "Faults&warnings"."Fault present" AND NOT "Functions"."Dosing function selected";
END_REGION

REGION Network 29: 1sec onshot
   RUNG wire#powerrail
      "R_TRIG_DB_16".R_TRIG(CLK := "Clock_1Hz", Q => "1sec_pulse")
   END_RUNG
   // the same network as SCL:
   "R_TRIG_DB_16"(CLK := "Clock_1Hz", Q => "1sec_pulse");   // R_TRIG
END_REGION

REGION Network 30: reset from site hmi pb pn
   RUNG wire#powerrail
      Contact( "reset pb" )
      wire#w1
      Coil( "Control"."reset from hmi _site_pb_PN" )
   END_RUNG
   RUNG wire#powerrail
      Contact( "Ack_hmi" )
      { S7_Templates := "time_type := Time" } "IEC_Timer_0_DB_21".TOF(pt := t#5s, et =>)
   END_RUNG wire#w1
   RUNG wire#powerrail
      Contact( "machine_on" )
      { S7_Templates := "time_type := Time" } "IEC_Timer_0_DB_20".TP(pt := t#1m, et =>)
   END_RUNG wire#w1
   // the same network as SCL:
   "IEC_Timer_0_DB_21".TOF(IN := "Ack_hmi", PT := t#5s);
   "IEC_Timer_0_DB_20".TP(IN := "machine_on", PT := t#1m);
   "Control"."reset from hmi _site_pb_PN" := "reset pb" OR "IEC_Timer_0_DB_21".Q OR "IEC_Timer_0_DB_20".Q;
END_REGION

REGION Network 31: pump maximum idle time in minutes
   RUNG wire#powerrail
      { S7_Templates := "SrcType := DInt" } Mul(in1 := "Control"."Pump A maximum Idle Time", in2 := 60000, out => "Control"."Pump A maximum Idle Time sec")
      { S7_Templates := "SrcType := DInt" } Mul(in1 := "Control"."Pump B maximum Idle Time", in2 := 60000, out => "Control"."Pump B maximum Idle Time sec")
   END_RUNG
   // the same network as SCL:
   "Control"."Pump A maximum Idle Time sec" := "Control"."Pump A maximum Idle Time" * 60000;
   "Control"."Pump B maximum Idle Time sec" := "Control"."Pump B maximum Idle Time" * 60000;
END_REGION

REGION Network 32: Mute
   RUNG wire#powerrail
      Contact( "buzzer" )
      Coil( "Control".Mute."Mute enable" )
   END_RUNG
   RUNG wire#powerrail
      Contact( "Control".Mute."Mute enable" )
      Contact( "Control".Mute."Mutte On" )
      S_Coil( "Control".Mute."Mute buzzer" )
   END_RUNG
   RUNG wire#powerrail
      Contact( "Control".Mute."Mute buzzer" )
      { S7_Templates := "time_type := Time" } "IEC_Timer_0_DB_94".TON(pt := T#5m, et =>)
      wire#w1
      R_Coil( "Control".Mute."Mute buzzer" )
   END_RUNG
   RUNG wire#powerrail
      I_Contact( "Faults&warnings"."Fault present" )
   END_RUNG wire#w1
   RUNG wire#w1
      R_Coil( "Control".Mute."Mutte On" )
   END_RUNG
   // the same network as SCL:
   "Control".Mute."Mute enable" := "buzzer";
   IF "Control".Mute."Mute enable" AND "Control".Mute."Mutte On" THEN
       "Control".Mute."Mute buzzer" := TRUE;
   END_IF;
   "IEC_Timer_0_DB_94".TON(IN := "Control".Mute."Mute buzzer", PT := T#5m);
   IF "IEC_Timer_0_DB_94".Q OR NOT "Faults&warnings"."Fault present" THEN
       "Control".Mute."Mute buzzer" := FALSE;
       "Control".Mute."Mutte On" := FALSE;
   END_IF;
END_REGION
END_FUNCTION
